Fanuc KAREL source: kt00637.KL

-- PROVISIONAL review KL for V770-1; original PC SHA256 08599f0989357e66cbd720ea4f244e7bea6bd99fe1744f468389d5617784ee86
-- Incomplete behavior may be omitted. Consult companion uncertainty JSON. Do not deploy.
PROGRAM KT00637
%NOLOCKGROUP
VAR
  OUT : INTEGER
-- UNRESOLVED_DECL Y1 type=002018
-- UNRESOLVED_DECL Y2 type=002018
BEGIN
  -- UNRESOLVED_PC offsets 5-19; opcodes 2E,22,9D,33,B2
  -- UNRESOLVED_PC offsets 24-38; opcodes 2E,22,9D,33,B2
  -- UNRESOLVED_PC offsets 43-57; opcodes 2E,22,9D,33,B2
  -- UNRESOLVED_PC offsets 62-76; opcodes 2E,22,9D,33,B2
  -- UNRESOLVED_PC offsets 81-96; opcodes 22,9D,33,B1,23
  -- UNRESOLVED_PC offsets 101-105; opcodes 7F
END KT00637
